// Mitsubishi GX Works2 project: intel7기 정성욱_스마트설비제어_평가   PLC: Q02/Q02H

PROGRAM MAIN
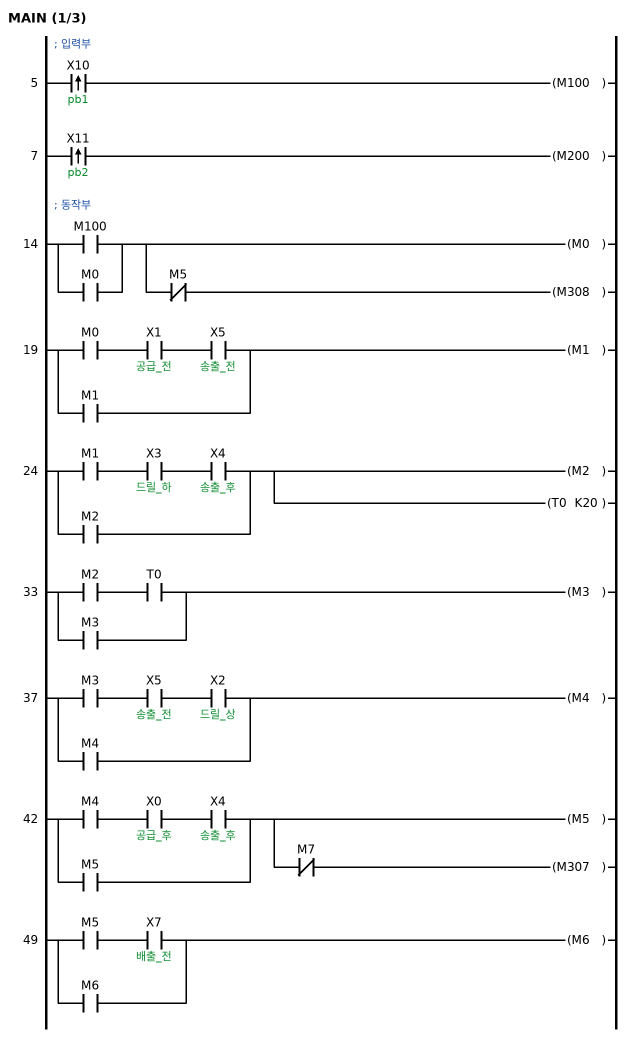
; 입력부
5     LDP     X10  ; pb1
      OUT     M100
7     LDP     X11  ; pb2
      OUT     M200
; 동작부
14    LD      M100
      OR      M0
      OUT     M0
      ANI     M5
      OUT     M308
19    LD      M0
      AND     X1  ; 공급_전
      AND     X5  ; 송출_전
      OR      M1
      OUT     M1
24    LD      M1
      AND     X3  ; 드릴_하
      AND     X4  ; 송출_후
      OR      M2
      OUT     M2
      OUT     T0 K20
33    LD      M2
      AND     T0
      OR      M3
      OUT     M3
37    LD      M3
      AND     X5  ; 송출_전
      AND     X2  ; 드릴_상
      OR      M4
      OUT     M4
42    LD      M4
      AND     X0  ; 공급_후
      AND     X4  ; 송출_후
      OR      M5
      OUT     M5
      ANI     M7
      OUT     M307
49    LD      M5
      AND     X7  ; 배출_전
      OR      M6
      OUT     M6
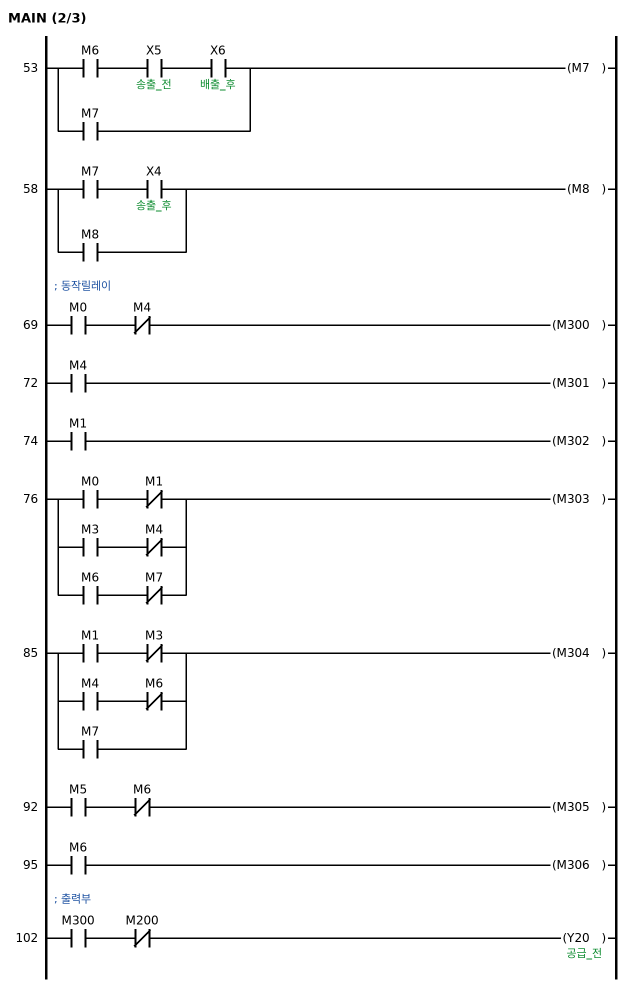
53    LD      M6
      AND     X5  ; 송출_전
      AND     X6  ; 배출_후
      OR      M7
      OUT     M7
58    LD      M7
      AND     X4  ; 송출_후
      OR      M8
      OUT     M8
; 동작릴레이
69    LD      M0
      ANI     M4
      OUT     M300
72    LD      M4
      OUT     M301
74    LD      M1
      OUT     M302
76    LD      M0
      ANI     M1
      LD      M3
      ANI     M4
      ORB
      LD      M6
      ANI     M7
      ORB
      OUT     M303
85    LD      M1
      ANI     M3
      LD      M4
      ANI     M6
      ORB
      OR      M7
      OUT     M304
92    LD      M5
      ANI     M6
      OUT     M305
95    LD      M6
      OUT     M306
; 출력부
102   LD      M300
      ANI     M200
      OUT     Y20  ; 공급_전
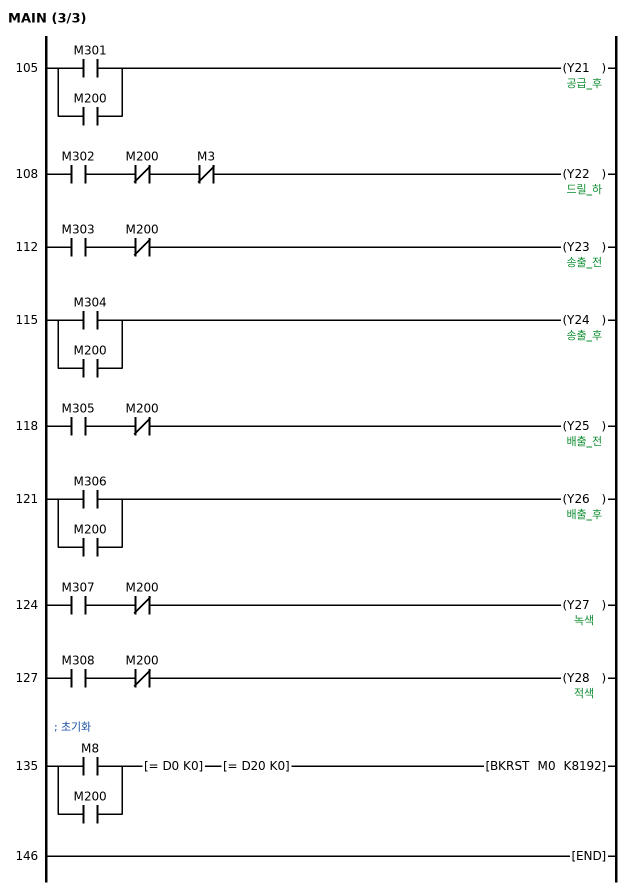
105   LD      M301
      OR      M200
      OUT     Y21  ; 공급_후
108   LD      M302
      ANI     M200
      ANI     M3
      OUT     Y22  ; 드릴_하
112   LD      M303
      ANI     M200
      OUT     Y23  ; 송출_전
115   LD      M304
      OR      M200
      OUT     Y24  ; 송출_후
118   LD      M305
      ANI     M200
      OUT     Y25  ; 배출_전
121   LD      M306
      OR      M200
      OUT     Y26  ; 배출_후
124   LD      M307
      ANI     M200
      OUT     Y27  ; 녹색
127   LD      M308
      ANI     M200
      OUT     Y28  ; 적색
; 초기화
135   LD      M8
      OR      M200
      AND=    D0 K0
      AND=    D20 K0
      BKRST   M0 K8192
146   END
END_PROGRAM

PROGRAM HMI
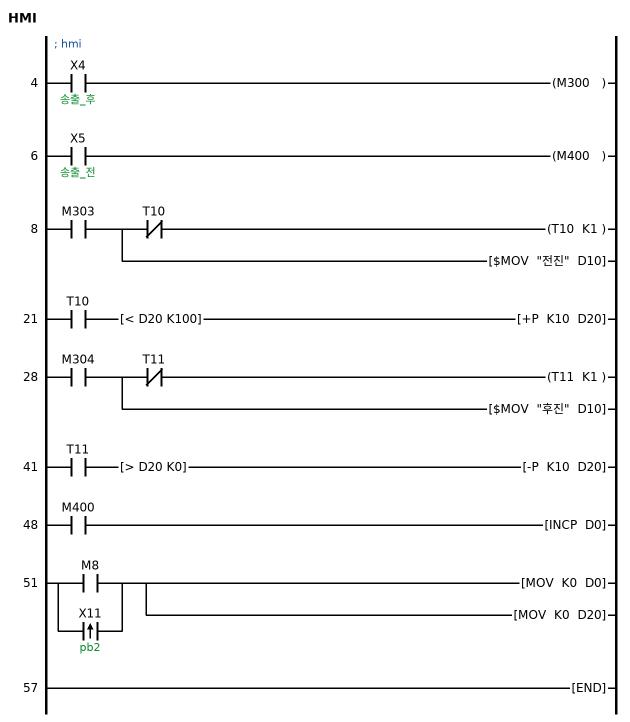
; hmi
4     LD      X4  ; 송출_후
      OUT     M300
6     LD      X5  ; 송출_전
      OUT     M400
8     LD      M303
      MPS
      ANI     T10
      OUT     T10 K1
      MPP
      $MOV    "전진" D10
21    LD      T10
      AND<    D20 K100
      +P      K10 D20
28    LD      M304
      MPS
      ANI     T11
      OUT     T11 K1
      MPP
      $MOV    "후진" D10
41    LD      T11
      AND>    D20 K0
      -P      K10 D20
48    LD      M400
      INCP    D0
51    LD      M8
      ORP     X11  ; pb2
      MOV     K0 D0
      MOV     K0 D20
57    END
END_PROGRAM

// device comments not shown above
X8  ; 매거진
X9  ; 비금속
X0A  ; 금속
X12  ; pb3
X13  ; pb4
X14  ; pb5
